Staubli VAL3: Axis8Action.pgx

public program Axis8Action(num x_nType (dimensions=1))
begin

  //七轴的IO动作

  switch x_nType

    //点动正
    case 1
      if dDio["O4_b8StopMotor"]==true
        dDio["O4_b8StopMotor"]=false
        delay(0.05)
      endIf
      dDio["O4_b8MoveDir"]=true
      //aioSet(aAio["O4_a8JogVelo"],50)
      delay(0.2)

    break

    //点动负
    case 2
      if dDio["O4_b8StopMotor"]==true
        dDio["O4_b8StopMotor"]=false
        delay(0.05)
      endIf
      dDio["O4_b8MoveDirM"]=true
      //  aioSet(aAio["O4_a8JogVelo"],50)
      delay(0.2)
    break

    //回到机械零位
    case 4
      dDio["O4_b8StopMotor"]=false
      dDio["O4_b8AxisHome"]=true
      delay(0.2)
    break





    //停止运动
    case 6
      dDio["O4_b8StopMotor"]=true
      delay(0.2)
      dDio["O4_b8StopMotor"]=false
    break


    case 6

    break


    //没有按钮按下
    case 9
      dDio["O4_b8ResetError"]=false
      dDio["O4_b8AxisHome"]=false
      dDio["O4_b8MoveDirM"]=false
      dDio["O4_b8MoveDir"]=false
    break


    //复位
    case 10
      dDio["O4_b8StopMotor"]=false
      dDio["O4_b8ResetError"]=true
      // dDio["O4_b8StopMotor"]=false
      delay(0.2)
    break
    default
    break

  endSwitch


end
